INTERFACE ITF_Node

METHOD GetLastNode : ITF_Node
VAR_INPUT
END_VAR
END_METHOD

METHOD GetMyPointer : PVOID
END_METHOD

METHOD GetNextNode : ITF_Node
VAR_INPUT
END_VAR
END_METHOD

METHOD GetPositionInList : UINT
VAR_INPUT
END_VAR
END_METHOD

METHOD SetLastNode : BOOL
VAR_INPUT
	Node	: ITF_Node;
END_VAR
END_METHOD

METHOD SetNextNode : BOOL
VAR_INPUT
	Node	: ITF_Node;
END_VAR
END_METHOD

METHOD SetPositionInList : BOOL
VAR_INPUT
	Index		: UINT;
END_VAR
END_METHOD

END_INTERFACE

(* stored: Version 1.1.0.1
   Itf ITF_Node: Id {ce730fea-0410-4f82-be09-48838bf80d7d}
   Method GetLastNode: Id {d049d641-fad6-4de4-940f-5381d88de601}
   Method GetMyPointer: Id {91ea8946-01ec-4f63-900f-b472806387f9}
   Method GetNextNode: Id {c50ec64b-e253-4640-a8c4-d08f97ec3a30}
   Method GetPositionInList: Id {40bf4a88-7fbd-4518-9f62-0d4880200513}
   Method SetLastNode: Id {16b6a02a-d638-456d-b67c-3f8cac31805a}
   Method SetNextNode: Id {25af4737-91ba-4cc5-b030-0922a7c4b529}
   Method SetPositionInList: Id {c27435fc-812e-464b-9e22-f1c5ef8a5103} *)
